FUNCTION_BLOCK FB_VisionSensor (* Capteur vision - detecte changement de couleur *)
  (* Standard: 61499-2 *)
  (* Version 2.0, 20/01/2026, Claude, Schneider Electric, Detecte si couleur change *)
  PACKAGE Main;
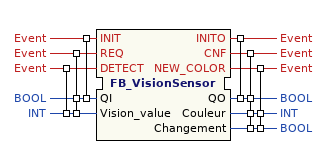
  EVENT_INPUT
    INIT WITH QI; (* Initialization Request *)
    REQ WITH QI, Vision_value; (* Normal Execution Request *)
    DETECT WITH Vision_value; (* Piece presente - lire couleur *)
  END_EVENT
  EVENT_OUTPUT
    INITO WITH QO; (* Initialization Confirm *)
    CNF WITH QO, Couleur, Changement; (* Execution Confirmation *)
    NEW_COLOR WITH Couleur, Changement; (* Nouvelle couleur detectee *)
  END_EVENT
  VAR_INPUT
    QI : BOOL; (* Input event qualifier *)
    Vision_value : INT; (* Valeur capteur vision (0-9) *)
  END_VAR
  VAR_OUTPUT
    QO : BOOL; (* Output event qualifier *)
    Couleur : INT; (* 0=Aucune, 1=Bleu, 2=Vert, 3=Gris *)
    Changement : BOOL; (* TRUE si couleur differente de la precedente *)
  END_VAR
  VAR
    Couleur_Precedente : INT; (* Couleur de la piece precedente *)
  END_VAR
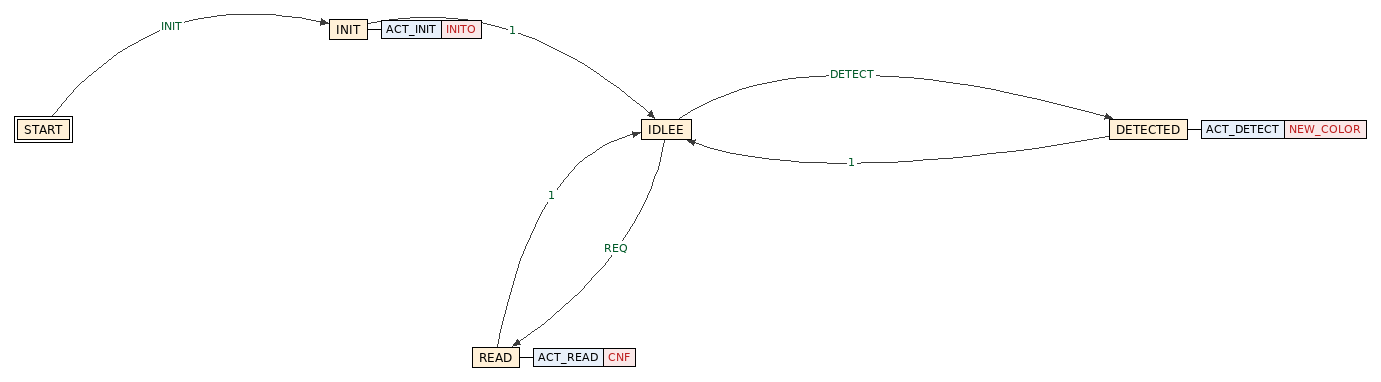
  EC_STATES
    START; (* Initial State *)
    INIT : ACT_INIT -> INITO; (* Initialization *)
    IDLEE; (* En attente *)
    READ : ACT_READ -> CNF; (* Lecture valeur *)
    DETECTED : ACT_DETECT -> NEW_COLOR; (* Piece detectee *)
  END_STATES
  EC_TRANSITIONS
    START TO INIT := INIT;
    INIT TO IDLEE := 1;
    IDLEE TO READ := REQ;
    READ TO IDLEE := 1;
    IDLEE TO DETECTED := DETECT;
    DETECTED TO IDLEE := 1;
  END_TRANSITIONS
  ALGORITHM ACT_INIT IN ST: (* Initialization *)
QO := TRUE;
Couleur := 0;
Changement := FALSE;
Couleur_Precedente := 0;
  END_ALGORITHM
  ALGORITHM ACT_READ IN ST: (* Lecture valeur capteur *)
(* Convertir Vision_value en Couleur *)
IF Vision_value > 0 AND Vision_value < 4 THEN
    Couleur := 1;  (* Bleu *)
ELSIF Vision_value >= 4 AND Vision_value < 7 THEN
    Couleur := 2;  (* Vert *)
ELSIF Vision_value >= 7 THEN
    Couleur := 3;  (* Gris *)
ELSE
    Couleur := 0;  (* Aucune piece *)
END_IF;
  END_ALGORITHM
  ALGORITHM ACT_DETECT IN ST: (* Piece detectee - comparer avec precedente *)
(* Convertir Vision_value en Couleur *)
IF Vision_value > 0 AND Vision_value < 4 THEN
    Couleur := 1;  (* Bleu *)
ELSIF Vision_value >= 4 AND Vision_value < 7 THEN
    Couleur := 2;  (* Vert *)
ELSIF Vision_value >= 7 THEN
    Couleur := 3;  (* Gris *)
ELSE
    Couleur := 0;  (* Aucune piece *)
END_IF;

(* Detecter si la couleur a change *)
IF Couleur_Precedente <> 0 AND Couleur <> Couleur_Precedente THEN
    Changement := TRUE;   (* Couleur DIFFERENTE de la precedente *)
ELSE
    Changement := FALSE;  (* Meme couleur OU premiere piece *)
END_IF;
Couleur_Precedente := Couleur;
  END_ALGORITHM
END_FUNCTION_BLOCK
